FUNCTION_BLOCK FB_ReadPM5350 EXTENDS ReadPm5350

VAR_OUTPUT
END_VAR
VAR PERSISTENT
	validEnvergyIntoLoad : LREAL;
END_VAR
(*VAR_IN_OUT
	PM		:	ST_PowerMeter;
END_VAR*)
VAR
	bOtherDataGood : BOOL;
END_VAR

SUPER^(PM:= THIS^.PM,
		bExecute := bExecute);

bOtherdataGood := 	IsGoodData( pm.Basic.Voltage_LLAvg )
				AND IsGoodData( pm.Basic.Current_Avg)
				AND IsGoodData(	pm.Basic.Frequency)
				AND IsGoodData( pm.Basic.Voltage_AN)
				AND IsGoodData(	pm.Basic.Voltage_AB)
				AND IsGoodData( pm.Basic.Voltage_BN)
				AND IsGoodData(	pm.Basic.Voltage_BC)
				AND IsGoodData( pm.Basic.Voltage_CN)
				AND IsGoodData(	pm.Basic.Voltage_CA);
				
				
IF IsGoodData (pm.Basic.RealEnergy_IntoLoad ) AND bOtherDataGood THEN
	;// pm.Basic.RealEnergy_IntoLoad still it
	validEnvergyIntoLoad := pm.Basic.RealEnergy_IntoLoad;
ELSE
	pm.Basic.RealEnergy_IntoLoad := validEnvergyIntoLoad;
END_IF

//round value
	(*PM.Basic.RealEnergy_IntoLoad := F_RoundLrealEx(	lrIn 	:= PM.Basic.RealEnergy_IntoLoad,
										iPrecision 	:= 0);*)
												
	PM.Basic.PowerFactor := F_RoundLrealEx(	lrIn 	:= PM.Basic.PowerFactor,
								iPrecision 	:= 2);

END_FUNCTION_BLOCK

(* stored: Version 1.1.0.1, ProductVersion 3.1.4024.12
   POU FB_ReadPM5350: Id {ba443878-5f2f-4215-8d9d-4bc7b40e7c5a}, SpecialFunc None *)
